FUNCTION F_PVOID_ARG : ST_Arg
VAR_INPUT
	pInput : PVOID;
END_VAR
VAR
	stArg : ST_Arg;
	sysVar_Info : __SYSTEM.VAR_INFO;
END_VAR

sysVar_Info 	:= __VARINFO(pInput);
stArg.TypeClass := sysVar_Info.TypeClass;
stArg.pValue 	:= pInput;
stArg.diSize 	:= SIZEOF(pInput);
stArg.sValue 	:= TO_STRING(pInput); 
F_PVOID_ARG := stArg;

END_FUNCTION

(* stored: Version 1.1.0.1, ProductVersion 3.1.4024.4
   POU F_PVOID_ARG: Id {702af97a-af11-41ab-adb0-d2e943093741}, SpecialFunc None *)
